Omron CX-Programmer project NewProject (CX-Programmer 9.51)

# PLC my_first_project: CP1L L
; Comment

## Program NewProgram1 (cyclic task 0)
Local symbols
button_1 0.00 BOOL
button_2 0.01 BOOL
button_3 0.02 BOOL
out_1 100.00 BOOL
out_2 100.01 BOOL

### Section Section1

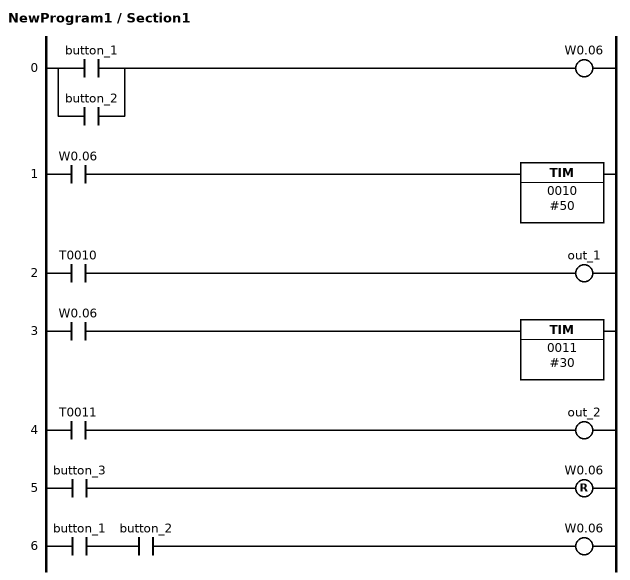
; rung 0
LD button_1
OR button_2
OUT W0.06
; rung 1
LD W0.06
TIM 0010 #50
; rung 2
LD T0010
OUT out_1
; rung 3
LD W0.06
TIM 0011 #30
; rung 4
LD T0011
OUT out_2
; rung 5
LD button_3
RSET W0.06
; rung 6
LD button_1
AND button_2
OUT W0.06

### Section END
; rung 0
END(001)